PROGRAM PRG_TEST_FB_PARAMETERHANDLER
VAR
	fbParameterHandler 	: FB_ParameterHandler;
	stParameterId		: Udt_ParameterId;
	stParameter 		: Udt_Parameter; // NOTE: Udt_Parameter is persistent
	bAddParameter 		: BOOL;
END_VAR

fbParameterHandler();

IF bAddParameter THEN
	bAddParameter := FALSE;
	fbParameterHandler.CmdAddParameter(stParameter);
END_IF

END_PROGRAM

(* stored: Version 1.1.0.1, ProductVersion 3.1.4024.11
   POU PRG_TEST_FB_PARAMETERHANDLER: Id {0c300e5c-bc84-0976-09ac-2d3645d53aac}, SpecialFunc None *)
